INTERFACE I_PackML_UnholdingCommands

METHOD PUBLIC Abort
VAR_INPUT
END_VAR
END_METHOD

METHOD StateComplete
VAR_INPUT
END_VAR
END_METHOD

METHOD PUBLIC Stop
VAR_INPUT
END_VAR
END_METHOD

END_INTERFACE

(* stored: Version 1.1.0.1, ProductVersion 3.1.4024.12
   Itf I_PackML_UnholdingCommands: Id {2ed69181-4160-0c5d-1d9d-bb7c14caa326}
   Method Abort: Id {4e7e3af3-28c7-0217-0911-25fd9ed0093f}
   Method StateComplete: Id {2e335044-0308-0546-193b-aceb6a225033}
   Method Stop: Id {4577b164-d5e6-028f-054b-5e25dcb4c9bc} *)
